(* IEC 61131-3 sources: teller/JD_Teller_LC2_V11/Class/VaranManagerPostScan, 1 file *)

(* ---- VaranManagerPostScan.st ---- *)
(*!
<Class
	Name               = "VaranManagerPostScan"
	Revision           = "1.1"
	RealtimeTask       = "false"
	CyclicTask         = "false"
	BackgroundTask     = "false"
	Sigmatek           = "true"
	OSInterface        = "false"
	HighPriority       = "true"
	Automatic          = "true"
	UpdateMode         = "Postscan"
	IconPath           = ".\Class\Tool.ico"
	SharedCommandTable = "true"
	Objectsize         = "(284,120)">
	<Channels>
		<Server Name="Server0" Visualized="true" Initialize="false" WriteProtected="true" Retentive="false"/>
		<Client Name="ManagerConnect" Required="true" Internal="false"/>
	</Channels>
</Class>
*)
VaranManagerPostScan : CLASS
  //Servers:
	Server0 	: SvrChCmd_DINT;
  //Clients:
	ManagerConnect 	: CltChCmd_VaranManager_Base;
  //Variables:
  //Functions:
				//! <Function Comment="[#ENGLISH]&#13;&#10;=================================================================================================&#13;&#10;Function to call CyWork() of VaranMaster&#13;&#10;=================================================================================================&#13;&#10;" Name="CyWork"/>
	FUNCTION VIRTUAL GLOBAL CyWork
		VAR_INPUT
			EAX 	: UDINT := EAX;
		END_VAR
		VAR_OUTPUT
			state (EAX) 	: UDINT;
		END_VAR;
  //Tables:
	FUNCTION @STD
		VAR_OUTPUT
			ret_code	: CONFSTATES;
		END_VAR;
	FUNCTION GLOBAL TAB @CT_;
END_CLASS;

#pragma usingLtd VaranManager_Base

(************************************************************************************
*
*	Class to call cywork() of VaranManager in Postscan
*	Created : Sigmatek	/	SR	/	March-April 2006
*	Changes :
*		1.0 => 1.1	/	28.11.2006
*			first library version
*		0.2 => 1.0	/	09.10.2006
*			initial version
*		0.1 => 0.2	/	13.06.2006
*			second testversion
*		0.0	=> 0.1	/	03.04.2006
*			first testversion for fair in Hannover
*
************************************************************************************)

//[#ENGLISH]
//=================================================================================================
//Function to call CyWork() of VaranMaster
//=================================================================================================
FUNCTION VIRTUAL GLOBAL VaranManagerPostScan::CyWork
VAR_INPUT
	EAX		: UDINT;
END_VAR
VAR_OUTPUT
	state		: UDINT;
END_VAR

	ManagerConnect.CyWork( 0 );			//call cywork() of VaranManager

	state:= READY;

END_FUNCTION //VIRTUAL GLOBAL VaranManagerPostScan::CyWork
